// TIA Portal V17 export
// export: Created 2025-03-05T07:59:08.4573498Z, ExportSetting WithDefaults, DisplayName Totally Integrated Automation Portal, DisplayVersion V17 Update 8, DisplayName TIA Portal Openness, DisplayVersion V17 Update 8, DisplayName TIA Portal Version Control Interface, DisplayVersion V17, DisplayName SINAMICS Startdrive Advanced, DisplayVersion V17 SP2, DisplayName SINAMICS Startdrive G110M, G120, G120C, G120D, G120P, G115D, DisplayVersion V17 SP2, DisplayName SINAMICS Startdrive G130, G150, S120, S150, SINAMICS MV, S210, DisplayVersion V17 SP2, DisplayName STEP 7 Professional, DisplayVersion V17 Update 8, DisplayName SINUMERIK ONE STEP 7 Toolbox, DisplayVersion V17 Update 12, DisplayName SINUMERIK 840D sl STEP 7 Toolbox, DisplayVersion V17 Update 12, DisplayName STEP 7 Safety, DisplayVersion V17 Update 6, DisplayName WinCC Advanced, DisplayVersion V17 Update 8
DATA_BLOCK "DB2710_U1_F3_GRIPPER"   // DB2710
{ DB_Accessible_From_OPC_UA := 'FALSE' }
AUTHOR : ETXETAR
VERSION : 1.0
// stored: AutoNumber false, DBAccessibleFromOPCUA false, DBAccessibleFromWebserver true, InstanceOfName FB2509_CYL_OPEN_CLOSE_FIX_CLADDING, InstanceOfType FB
"FB2509_CYL_OPEN_CLOSE_FIX_CLADDING"
   // VAR_INPUT
   //    OPTIONS_0 : Byte;
   //    OPTIONS_1 : Byte;
   //    OPTIONS_2 : Byte;
   //    CLOSED_PART_A : Bool;
   //    CLOSED_PART_B : Bool;
   //    CLOSED_PART_C : Bool;
   //    CLOSED_PART_D : Bool;
   //    OPEN_PART_A : Bool;
   //    OPEN_PART_B : Bool;
   //    OPEN_PART_C : Bool;
   //    OPEN_PART_D : Bool;
   //    CLOSED_PRESSURE_SWITCH_1 : Bool;
   //    CLOSED_PRESSURE_SWITCH_2 : Bool;
   //    OPEN_PRESSURE_SWITCH_1 : Bool;
   //    OPEN_PRESSURE_SWITCH_2 : Bool;
   //    CLOSED_LOW_PRESSURE_SWITCH : Bool;
   //    OPEN_LOW_PRESSURE_SWITCH : Bool;
   //    GENERAL_CONDITIONS : Bool;
   //    CLOSE_CONDITIONS : Bool;
   //    OPEN_CONDITIONS : Bool;
   //    RELEASE_PRESSURE_CONDITIONS : Bool;
   //    LOW_PRESSURE_CONDITIONS : Bool;
   //    HYDRAULIC_OR_PNEUMATIC : Bool;
   //    FIXTURE_PART_TYPE_SEL : Bool;
   //    HMI_CMM_LINE_ACT_DEACT : Bool;
   //    HMI_CMM_LINE_RELEASE_LOW : Bool;
   //    HMI_CLOSE_MAN_REQ : Bool;
   //    HMI_OPEN_MAN_REQ : Bool;
   //    HMI_RELEASE_PRESSURE_MAN_REQ : Bool;
   //    HMI_LOW_PRESSURE_MAN_REQ : Bool;
   //    FLOWMETER_RESET : Bool;
   //    CLOSE_AUTO_REQ : Bool;
   //    OPEN_AUTO_REQ : Bool;
   //    RELEASE_PRESSURE_AUTO_REQ : Bool;
   //    LOW_PRESSURE_AUTO_REQ : Bool;
   //    M_VERIFY_CLOSED : Bool;
   //    M_VERIFY_OPEN : Bool;
   //    M_VERIFY_LOW_PRESSURE : Bool;
   //    CHECK_CLOSED_CNC_PLC_SIGNAL : Bool;
   //    CHECK_OPEN_CNC_PLC_SIGNAL : Bool;
   //    CHECK_CLOSED_LOW_PRESSURE_CNC_PLC_SIGNAL : Bool;
   //    CHECK_OPEN_LOW_PRESSURE_CNC_PLC_SIGNAL : Bool;
   //    CLOSE_FLOW_ACTIVE : Bool;
   //    UNIT_ALARM : UInt;
   //    STATION_ALARM : UInt;
   // END_VAR
   // VAR_OUTPUT
   //    CLOSED : Bool;
   //    OPEN_STATUS : Bool;
   //    PRESSURE_RELEASED : Bool;
   //    LOW_PRESSURED : Bool;
   //    HMI_MOTION_EXECUTABILITY_LEFT : Bool;
   //    HMI_MOTION_EXECUTABILITY_RIGHT : Bool;
   //    HMI_MOTION_EXECUTABILITY_LEFT_2 : Bool;
   //    HMI_MOTION_EXECUTABILITY_RIGHT_2 : Bool;
   //    HMI_MOTION_END_POS_LEFT : Bool;
   //    HMI_MOTION_END_POS_RIGHT : Bool;
   //    HMI_MOTION_END_POS_LEFT_2 : Bool;
   //    HMI_MOTION_END_POS_RIGHT_2 : Bool;
   //    HMI_MOTION_ACTIVE_LEFT : Bool;
   //    HMI_MOTION_ACTIVE_RIGHT : Bool;
   //    HMI_MOTION_ACTIVE_LEFT_2 : Bool;
   //    HMI_MOTION_ACTIVE_RIGHT_2 : Bool;
   //    ALARMS : "CYL_ALARMS_OPN_CLS";
   //    RESET_FLOWMETER : Bool;
   //    CLOSE : Bool;
   //    OPEN_ACTION : Bool;
   //    LOW_PRESSURE : Bool;
   //    SAFETY_UNBLOCK : Bool;
   //    PRESSURIZE_A : Bool;
   //    PRESSURIZE_B : Bool;
   //    PRESSURIZE_C : Bool;
   // END_VAR
   // VAR_IN_OUT
   //    OPEN_FLOW_ACTIVE_FLOWMETER : Bool;
   // END_VAR
   // VAR RETAIN
   //    CYL { S7_SetPoint := 'True'} : "OPEN_CLOSE";
   //    TIMER_CLOSED { S7_SetPoint := 'True'} : TON_TIME;
   //    TIMER_OPEN { S7_SetPoint := 'True'} : TON_TIME;
   //    TIMER_PRESSURE_RELEASED { S7_SetPoint := 'True'} : TON_TIME;
   //    TIMER_LOW_PRESSURE { S7_SetPoint := 'True'} : TON_TIME;
   //    TIMER_SIMULTANEITY { S7_SetPoint := 'True'} : TON_TIME;
   //    TIMER_TIME_EXCEEDED { S7_SetPoint := 'True'} : TON_TIME;
   //    TIMER_ACTD_PRESSURE_TIME_EXCEEDED_1 { S7_SetPoint := 'True'} : TON_TIME;
   //    TIMER_ACTD_PRESSURE_SWITCH_1 { S7_SetPoint := 'True'} : TON_TIME;
   //    "TIMER_ACTD PRESSURE_TIME_EXCEEDED_2" { S7_SetPoint := 'True'} : TON_TIME;
   //    "TIMER_ACTD PRESSURE_SWITCH_2" { S7_SetPoint := 'True'} : TON_TIME;
   //    TIMER_DEACTD_PRESSURE_TIME_EXCEEDED_1 { S7_SetPoint := 'True'} : TON_TIME;
   //    TIMER_DEACTD_PRESSURE_SWITCH_1 { S7_SetPoint := 'True'} : TON_TIME;
   //    TIMER_DEACTD_PRESSURE_TIME_EXCEEDED_2 { S7_SetPoint := 'True'} : TON_TIME;
   //    TIMER_DEACTD_PRESSURE_SWITCH_2 { S7_SetPoint := 'True'} : TON_TIME;
   //    TIMER_ACTD_LOW_PRESSURE_TIME_EXCEEDED { S7_SetPoint := 'True'} : TON_TIME;
   //    TIMER_ACTD_LOW_PRESSURE_SWITCH { S7_SetPoint := 'True'} : TON_TIME;
   //    TIMER_DEACTD_LOW_PRESSURE_TIME_EXCEEDED { S7_SetPoint := 'True'} : TON_TIME;
   //    TIMER_DEACTD_LOW_PRESSURE_SWITCH { S7_SetPoint := 'True'} : TON_TIME;
   //    TIMER_SAFETY_UNBLOCK { S7_SetPoint := 'True'} : TOF_TIME;
   //    TIMER_CLMP_RCVRY_CLAMPED { S7_SetPoint := 'True'} : TON_TIME;
   //    TIMER_CLMP_RCVRY_UNCLAMPED { S7_SetPoint := 'True'} : TON_TIME;
   // END_VAR
BEGIN
END_DATA_BLOCK
